PROGRAM MAIN
VAR
	RoomData : stRoomData;
END_VAR

Hardware_Simulation();

RoomData.Temperature := INT_TO_REAL(IO.hwAirDataIN.CH1) / 32767 * 50.0; // as 0-10V~0-32767~0-50°C
RoomData.Humidity := INT_TO_REAL(IO.hwAirDataIN.CH2) / 32767 * 100.0; // as 0-10V~0-32767~0-100%
RoomData.VOC := INT_TO_REAL(IO.hwAirDataIN.CH3) / 32767 * 100.0; // as 0-10V~0-32767~0-100%
RoomData.CO2 := INT_TO_REAL(IO.hwAirDataIN.CH4) / 32767 * 5000.0; // as 0-10V~0-32767~0-5000ppm

END_PROGRAM

(* stored: Version 1.1.0.1, ProductVersion 3.1.4024.2
   POU MAIN: Id {6bff2563-8138-4968-9328-b38d21e7b1ab}, SpecialFunc None *)
